Staubli VAL3: isFound.pgx

public program isFound(string& x_sName[], bool& x_bFound[])
  local num i
  local num j
  local num l_nSize[3]
  local string l_sString
  local num k
  local num l_nResult
  local string l_sEmpty
  local num l_nID
begin
  //
  // find if a program is inside the processList
  //
  x_bFound=false
  //
  // update
  //
  l_sEmpty=""
  call use:stringCopy(l_sEmpty,sProcessList)
  // check all
  call loadProcessList(l_nResult)
  // get the size of the three processList
  for i=0 to 2
    call getSize(l_nSize[i],i)
    // look in all the program
    for j=0 to max(l_nSize[i]-1,0)
      l_nID=0
      call getCycle(l_sString,l_nID,l_nID,j,i)
      if l_sString==x_sName
        x_bFound=true
        x_sName=l_sString
        return
      endIf
    endFor
  endFor
end
